PROGRAM commandDecoder
VAR
	command 	: STRING(255);
	Head_Loaded : STRING;
	index 		: INT := 0;
	
	actualX 	: LREAL;
	actualY 	: LREAL;
	actualZ 	: Lreal;
	
	wait100ms : TON;
	wait200ms : TON;
	
END_VAR

wait100ms(IN := COM.bEnable OR gvl.StopALL, pt := T#500MS);
wait200ms(IN := COM.bEnable OR gvl.StopALL, pt := T#1S);

IF ( NOT (com.sendCommand = '') ) THEN
	command := F_ToLCase(com.sendCommand);
	com.sendCommand := '';
END_IF

CASE index OF
	0:	//commands
		COM.bEnable := FALSE;
		COM.bCouple := FALSE;
		COM.bHome 	:= FALSE;
		COM.inUSe 	:= FALSE;
		
		IF ( NOT (command = '') ) THEN
			IF 		(command = 'error' OR com.IFerror) THEN		index := 999;
			ELSIF 	(command = 'reset') THEN					index := 10;
			ELSIF 	(command = 'stop') THEN						index := 20;
			ELSIF 	(command = 'do homing') THEN				index := 100;
			ELSIF 	(command = 'z to zero') THEN				index := 110;
			ELSIF 	(command = 'go xyz') THEN					index := 200;
			ELSIF 	(command = 'go xy') THEN					index := 205;
			ELSIF 	(command = 'x-axis') THEN					index := 210;
			ELSIF 	(command = 'y-axis') THEN					index := 220;
			ELSIF 	(command = 'z-axis') THEN					index := 230;
			ELSIF 	(command = 'exec gcode') THEN				index := 250;
			ELSIF 	(command = 'execute trace') THEN			index := 260;
			ELSIF 	(command = 'execute sort') THEN				index := 270;
			ELSIF 	(command = 'execute drill') THEN			index := 280;
			ELSIF 	(command = 'read position') THEN			index := 300;
			ELSIF 	(command = 'up') THEN						index := 450;
			ELSIF 	(command = 'down') THEN						index := 460;
			ELSIF 	(command = 'show object') THEN				index := 600;
			ELSE												index := 0;
			END_IF;
			command := '';
		ELSE 
			index := 0;
		END_IF;
		
	10:  //reset
		GVL.message_pub  := '{"text": "Resetting"}';
		GVL.bSendMessage := TRUE;
	
		gcode.bReset := TRUE;
		COM.bReset 	:= TRUE;
		COM.bEnable := FALSE;
		COM.bCouple := FALSE;
		COM.bHome 	:= FALSE;
		COM.inUSe 	:= FALSE;
		COM.bMoveX 	:= FALSE;
		COM.bMoveY 	:= FALSE;
		COM.bMoveZ 	:= FALSE;
		COM.bReset 	:= FALSE;	
		gcode.bReset := FALSE;
		
		index 		:= 0;
		
	20:  //Stop
		gvl.StopALL := TRUE;
		
		GVL.message_pub  := '{"text": "Stopping program"}';
		GVL.bSendMessage := TRUE;
		
		IF wait100ms.q THEN
			gvl.StopALL := FALSE;
			index 		:= 0;
		END_IF
			
	100: //Do homing
		COM.bEnable := TRUE;
		COM.bCouple := TRUE;
		COM.bHome 	:= TRUE;
		
		GVL.message_pub  := '{"text": "Doing homing"}';
		GVL.bSendMessage := TRUE;
		
		IF COM.bHomeBusy THEN
			COM.inUSe 	:= TRUE;
		ELSE
			COM.inUSe 	:= FALSE;
		END_IF
		IF COM.bHomeDone THEN
			COM.bEnable := FALSE;
			COM.bCouple := FALSE;
			COM.bHome 	:= FALSE;
			COM.inUSe 	:= FALSE;
			gvl.configHoming := TRUE;
			index 	:= 0;
		END_IF
		
	110: //set Z position to zero
		COM.bSetZ 		:= TRUE;
		
		GVL.message_pub  := '{"text": "Z axis has been set to zero"}';
		GVL.bSendMessage := TRUE;
		
		IF (COM.PosZ = 0 AND COM.bValid) THEN
			COM.bSetZ 	:= FALSE;
			gvl.configZaxis := TRUE;
			index 		:= 0;
		END_IF
				
	200: //Go to xyz Pos
    	COM.absX := (COM.goX);
		COM.absY := (COM.goY);
		COM.absZ := (COM.goZ);
		
		IF gvl.configHoming THEN
			COM.bEnable := TRUE;
			COM.bCouple := TRUE;
			
			IF wait100ms.Q THEN 
				COM.bMoveX 	:= TRUE;
				COM.bMoveY 	:= TRUE;
				COM.bMoveZ 	:= TRUE;
			END_IF

			IF COM.bMoveBusy THEN
				COM.inUSe 	:= TRUE;
			ELSE
				COM.inUSe 	:= FALSE;
			END_IF
			
			IF COM.bMoveDone THEN
				COM.bEnable := FALSE;
				COM.bCouple := FALSE;
				COM.inUSe 	:= FALSE;
				COM.bMoveX 	:= FALSE;
				COM.bMoveY 	:= FALSE;
				COM.bMoveZ 	:= FALSE;
				index 	:= 0;
			END_IF
		ELSE
			index 	:= 995;
		END_IF
		
	205: //Go to xy Pos
    	COM.absX := (COM.goX);
		COM.absY := (COM.goY);
		
		IF gvl.configHoming THEN
			COM.bEnable := TRUE;
			COM.bCouple := TRUE;
			
			IF wait100ms.Q THEN 
				COM.bMoveX 	:= TRUE;
				COM.bMoveY 	:= TRUE;
			END_IF
			
			IF COM.bMoveBusy THEN
				COM.inUSe 	:= TRUE;
			ELSE
				COM.inUSe 	:= FALSE;
			END_IF
			
			IF COM.bMoveXDone AND COM.bMoveYDone THEN
				COM.bEnable := FALSE;
				COM.bCouple := FALSE;
				COM.inUSe 	:= FALSE;
				COM.bMoveX 	:= FALSE;
				COM.bMoveY 	:= FALSE;
				COM.bMoveZ 	:= FALSE;
				index 	:= 0;
			END_IF
		ELSE
			index 	:= 995;
		END_IF
		
	210: //Go X Pos
	    COM.absX := (com.goX);
		
		IF gvl.configHoming THEN
			COM.bEnable := TRUE;
			COM.bCouple := TRUE;
		
			IF wait100ms.Q THEN 
				COM.bMoveX 	:= TRUE;
			END_IF
			
			IF COM.bMoveBusy THEN
				COM.inUSe 	:= TRUE;
			ELSE
				COM.inUSe 	:= FALSE;
			END_IF
			
			IF COM.bMoveXDone THEN
				COM.bEnable := FALSE;
				COM.bCouple := FALSE;
				COM.inUSe 	:= FALSE;
				COM.bMoveX 	:= FALSE;
				index 	:= 0;
			END_IF
		ELSE
			index 	:= 995;
		END_IF
		
	220: //Go Y Pos
		COM.absY := (com.goY);
		
		IF gvl.configHoming THEN
			COM.bEnable := TRUE;
			
			IF wait100ms.Q THEN 
				COM.bMoveY 	:= TRUE;
			END_IF
					
			IF COM.bMoveBusy THEN
				COM.inUSe 	:= TRUE;
			ELSE
				COM.inUSe 	:= FALSE;
			END_IF
			
			IF COM.bMoveYDone THEN
				COM.bEnable := FALSE;
				COM.bCouple := FALSE;
				COM.inUSe 	:= FALSE;
				COM.bMoveY 	:= FALSE;
				index 	:= 0;
			END_IF
		ELSE
			index 	:= 995;
		END_IF
			
	230: //Go Z Pos
		COM.absZ := (com.goZ);
		
		IF gvl.configZaxis THEN
			COM.bEnable := TRUE;
			
			IF wait100ms.Q THEN 
				COM.bMoveZ 	:= TRUE;
			END_IF
			
			IF COM.bMoveBusy THEN
				COM.inUSe 	:= TRUE;
			ELSE
				COM.inUSe 	:= FALSE;
			END_IF
			
			IF COM.bMoveZDone THEN
				COM.bEnable := FALSE;
				COM.bCouple := FALSE;
				COM.inUSe 	:= FALSE;
				COM.bMoveZ 	:= FALSE;
				index 	:= 0;
			END_IF
		ELSE
			index := 996;
		END_IF
		
	250: //Execute Gcode
		GVL.message_pub  := '{"text": "Executing code say reset after the program"}';
		GVL.bSendMessage := TRUE;
		
		IF gvl.configHoming AND FALSE THEN
			COM.bEnable := TRUE;
			gcode.bBuildGroup := TRUE;
			gcode.bLoad := TRUE;
						
			IF wait100ms.Q THEN 
				gcode.bStart 	:= TRUE;
				gcode.bLoad := FALSE;
			ELSE 
				gcode.bStart 	:= FALSE;
			END_IF
			
			IF 	(command = 'reset' OR command = 'stop') THEN
				gcode.bStop	:= TRUE;
				gcode.bReset := TRUE;
				gcode.bBuildGroup := FALSE;
				COM.bEnable := FALSE;
				
			ELSIF(gcode.bStop)THEN
					gcode.bStop	:= FALSE;
					gcode.bReset := FALSE;
					COM.bEnable := FALSE;
					
					index 		:= 0;
			END_IF
			
		ELSE
			index := 995;
		END_IF
			
	260: //execute trace
		GVL.message_pub  := '{"text": "Tracing will be executed"}';
		GVL.bSendMessage := TRUE;
		index 		:= 0;
		
	270: //execute sort
		GVL.message_pub  := '{"text": "executing sort"}';
		GVL.bSendMessage := TRUE;
		index 		:= 0;
		
	280: //execute drill
		GVL.message_pub  := '{"text": "execute drill"}';
		GVL.bSendMessage := TRUE;
		index 		:= 0;
		
	300: //Read XYZ
		actualX 	:= COM.PosX;
		actualY 	:= COM.Posy;
		actualZ 	:= COM.PosZ;
		IF COM.bValid THEN
			index 	:= 0;
		END_IF
	
	450: //Up
		COM.relZ := (-com.goZ);
		COM.bEnable := TRUE;
		
		IF wait100ms.Q THEN 
			COM.bRelZ 	:= TRUE;
		END_IF
		
		IF COM.bMoveBusy THEN
			COM.inUSe 	:= TRUE;
		ELSE
			COM.inUSe 	:= FALSE;
		END_IF
		
		IF COM.bMoveZRelDone THEN
			COM.bEnable := FALSE;
			COM.bCouple := FALSE;
			COM.inUSe 	:= FALSE;
			COM.brelZ 	:= FALSE;
			index 	:= 0;
		END_IF	
	
	460: //Down
		COM.relZ := (com.goZ);
		COM.bEnable := TRUE;
		
		IF wait100ms.Q THEN 
			COM.bRelZ 	:= TRUE;
		END_IF
		
		IF COM.bMoveBusy THEN
			COM.inUSe 	:= TRUE;
		ELSE
			COM.inUSe 	:= FALSE;
		END_IF
		
		IF COM.bMoveZRelDone THEN
			COM.bEnable := FALSE;
			COM.bCouple := FALSE;
			COM.inUSe 	:= FALSE;
			COM.brelZ 	:= FALSE;
			index 	:= 0;
		END_IF
			
	600: //Show object
		com.objectNum := com.object1;
		com.readfile  := TRUE;

		
		IF gvl.configHoming THEN
			COM.bEnable := TRUE;
			COM.bCouple := TRUE;
			
			IF wait100ms.Q THEN 
				COM.absX := LREAL_TO_INT(COM.objectx);
				COM.absY := LREAL_TO_INT(COM.objecty);
				com.objectread := TRUE;
			END_IF
			
			IF wait200ms.Q THEN 
				COM.bMoveX 	:= TRUE;
				COM.bMoveY 	:= TRUE;
				com.objectread := FALSE;
			END_IF
			
			IF COM.bMoveBusy THEN
				COM.inUSe 	:= TRUE;
			ELSE
				COM.inUSe 	:= FALSE;
			END_IF
			
			IF COM.bMoveXDone AND COM.bMoveYDone THEN
				COM.bEnable := FALSE;
				COM.bCouple := FALSE;
				COM.inUSe 	:= FALSE;
				COM.bMoveX 	:= FALSE;
				COM.bMoveY 	:= FALSE;
				COM.bMoveZ 	:= FALSE;
				index 	:= 0;
			END_IF
		ELSE
			index 	:= 995;
		END_IF
	

	996: //set z to zero before performing an action on the z axis
		GVL.message_pub  := '{"text": "You have to do Z to zero first"}';
		GVL.bSendMessage := TRUE;
		index := 0;
	999: //Error
			COM.bEnable := FALSE;
			gvl.StopALL := TRUE;
			GVL.message_pub  := '{"text": "There has been an error use reset command"}';
			GVL.bSendMessage := TRUE;
			IF(command = 'reset')THEN
				gvl.StopALL := FALSE;
				index := 0;
			END_IF

	ELSE 
		index := 0;
END_CASE;

END_PROGRAM

(* stored: Version 1.1.0.1, ProductVersion 3.1.4024.2
   POU commandDecoder: Id {7eba7217-46bb-46ef-8690-bb184ce360f6}, SpecialFunc None *)
